TYPE DM430GNScreenConfig EXTENDS DeviceConfiguration :
STRUCT
	SerialCommunication : SerialCommunication;
END_STRUCT
END_TYPE

(* stored: Version 1.1.0.1, ProductVersion 3.1.4024.12
   DUT DM430GNScreenConfig: Id {1a8f042e-b2b1-4845-9d52-4df4a237bd7e} *)
